// TwinCAT 3 PLC project PLC1
// ProgramVersion: 3.1.4023.0
// libraries:
//   Tc2_Standard, * (Beckhoff Automation GmbH)
//   Tc2_System, * (Beckhoff Automation GmbH)
//   Tc3_Module, * (Beckhoff Automation GmbH)
// project tree:
//   / PlcTask.TcTTO
//   POUs/ MAIN.TcPOU
//   POUs/SD_Valve/ SD_Valve.TcPOU
//   POUs/SD_Valve/States/ InitState.TcPOU, AutoState.TcPOU, ManualState.TcPOU, I_SD_ValveState.TcIO
//   POUs/SD_Valve/Transitions/ GoToManual.TcPOU, GoToInit.TcPOU, GoToAuto.TcPOU, I_Transitive.TcIO
// real-time tasks:
//   TASK PlcTask: cycle T#10ms, priority 20, ADS port 350

CONFIGURATION PLC1
    RESOURCE PLC ON TwinCAT3
        TASK PlcTask(INTERVAL := T#10ms, PRIORITY := 20);
        PROGRAM MAIN WITH PlcTask : MAIN;
    END_RESOURCE
END_CONFIGURATION

// ---- POUs/SD_Valve/States/I_SD_ValveState.TcIO
INTERFACE I_SD_ValveState

METHOD Close : BOOL
VAR_INPUT
END_VAR
END_METHOD

METHOD Open : BOOL
VAR_INPUT
END_VAR
END_METHOD

METHOD RUN
END_METHOD

METHOD SetTransition
VAR_INPUT
    transition : I_Transitive;
END_VAR
END_METHOD

PROPERTY StateName : STRING
GET
END_GET
END_PROPERTY

END_INTERFACE

// ---- POUs/SD_Valve/Transitions/I_Transitive.TcIO
INTERFACE I_Transitive

METHOD Transit
VAR_INPUT
END_VAR
END_METHOD

END_INTERFACE

// ---- POUs/MAIN.TcPOU
PROGRAM MAIN
VAR
    sdValve : SD_Valve;
    openCmd : BOOL;
    openResult : BOOL;
    closeCmd : BOOL;
    closeResult : BOOL;
    goToAutoCmd : BOOL;
    goToManaulCmd : BOOL;
    goToInitCmd : BOOL;
END_VAR

sdValve();

IF openCmd THEN
    openCmd := FALSE;
    openResult := FALSE;
    openResult :=sdValve.OpenValve();
END_IF

IF closeCmd THEN
    closeCmd := FALSE;
    closeResult := FALSE;
    closeResult := sdValve.CloseValve();
END_IF

IF goToAutoCmd THEN
    goToAutoCmd := FALSE;
    sdValve.GoToAutoState();
END_IF

IF goToManaulCmd THEN
    goToManaulCmd := FALSE;
    sdValve.GoToManualState();
END_IF

IF goToInitCmd THEN
    goToInitCmd := FALSE;
    sdValve.GoToInitState();
END_IF

END_PROGRAM

// ---- POUs/SD_Valve/SD_Valve.TcPOU
FUNCTION_BLOCK SD_Valve
VAR_INPUT
END_VAR
VAR_OUTPUT
    coil : BOOL;
END_VAR
VAR
    _initState : InitState(THIS);
    _autoState : AutoState(THIS);
    _manualState : ManualState(THIS);
    _state : I_SD_ValveState := _initState;
    _stateName : STRING;
    _goToInit : GoToInit(ADR(_state), _initState);
    _goToAuto : GoToAuto(ADR(_state), _autoState);
    _goToManual : GoToManual(ADR(_state), _manualState);
    _setDefaultTransitions : BOOL := TRUE;
END_VAR

IF _setDefaultTransitions THEN
    _setDefaultTransitions := FALSE;
    _initState.SetTransition(_goToAuto);
END_IF

_state.RUN();
_stateName := _state.StateName;

METHOD CloseValve : BOOL
CloseValve := _state.Close();
END_METHOD

METHOD GoToAutoState
IF _state.StateName = _autoState.StateName THEN
    RETURN;
END_IF

IF _state.StateName = _initState.StateName THEN
    _state.SetTransition(_goToAuto);
ELSE
    _goToInit.Transit();
END_IF
END_METHOD

METHOD GoToInitState
IF _state.StateName = _initState.StateName THEN
    RETURN;
END_IF

_goToInit.Transit();
END_METHOD

METHOD GoToManualState
IF _state.StateName = _manualState.StateName THEN
    RETURN;
END_IF

IF _state.StateName = _initState.StateName THEN
    _state.SetTransition(_goToManual);
ELSE
    _goToManual.Transit();
END_IF
END_METHOD

METHOD OpenValve : BOOL
OpenValve := _state.Open();
END_METHOD

END_FUNCTION_BLOCK

// ---- POUs/SD_Valve/States/InitState.TcPOU
FUNCTION_BLOCK InitState IMPLEMENTS I_SD_ValveState
VAR_INPUT
END_VAR
VAR_OUTPUT
END_VAR
VAR
    _ptSdValve : POINTER TO SD_Valve;
    _transition : I_Transitive;
    delayTimer : Tc2_Standard.TON;
    start : BOOL;
END_VAR

delayTimer(IN:=start,PT:=T#10S);
IF NOT start THEN
    start := TRUE;
END_IF
IF delayTimer.q THEN
    start := FALSE;
//    _ptSdValve^.GoToAutoState();
    IF _transition<>0 THEN
        _transition.Transit();
	END_IF
END_IF

METHOD Close : BOOL
Close := false;
END_METHOD

METHOD FB_init : BOOL
VAR_INPUT
	bInitRetains : BOOL; // if TRUE, the retain variables are initialized (warm start / cold start)
	bInCopyCode : BOOL;  // if TRUE, the instance afterwards gets moved into the copy code (online change)
    ptSdValve : POINTER TO SD_Valve;
END_VAR
_ptSdValve := ptSdValve;
END_METHOD

METHOD Open : BOOL
Open := False;
END_METHOD

METHOD RUN
THIS^();
END_METHOD

METHOD SetTransition
VAR_INPUT
	transition	: I_Transitive;
END_VAR
_transition := transition;
END_METHOD

PROPERTY StateName : STRING
GET
StateName := 'Init';
END_GET
END_PROPERTY

END_FUNCTION_BLOCK

// ---- POUs/SD_Valve/States/AutoState.TcPOU
FUNCTION_BLOCK AutoState IMPLEMENTS I_SD_ValveState
VAR_INPUT
END_VAR
VAR_OUTPUT
END_VAR
VAR
    _ptSdValve : POINTER TO SD_Valve;
    _transition : I_Transitive;
END_VAR

METHOD Close : BOOL
Close := TRUE;
END_METHOD

METHOD FB_init : BOOL
VAR_INPUT
	bInitRetains : BOOL; // if TRUE, the retain variables are initialized (warm start / cold start)
	bInCopyCode : BOOL;  // if TRUE, the instance afterwards gets moved into the copy code (online change)
    ptSdValve : POINTER TO SD_Valve;
END_VAR
_ptSdValve := ptSdValve;
END_METHOD

METHOD Open : BOOL
Open := true;
END_METHOD

METHOD RUN
THIS^();
END_METHOD

METHOD SetTransition
VAR_INPUT
	transition	: I_Transitive;
END_VAR
_transition := transition;
END_METHOD

PROPERTY StateName : STRING
GET
StateName := 'Auto';
END_GET
END_PROPERTY

END_FUNCTION_BLOCK

// ---- POUs/SD_Valve/States/ManualState.TcPOU
FUNCTION_BLOCK ManualState IMPLEMENTS I_SD_ValveState
VAR_INPUT
END_VAR
VAR_OUTPUT
END_VAR
VAR
    _ptSdValve : POINTER TO SD_Valve;
    _transition : I_Transitive;
    delayTimer : Tc2_Standard.TP;
    command : BOOL;
END_VAR

delayTimer(IN:=command,PT:=T#5S);
IF command THEN
    command := FALSE;
END_IF

METHOD Close : BOOL
IF delayTimer.Q THEN
    Close := FALSE;
ELSE
    command := TRUE;
    Close := TRUE;
END_IF
END_METHOD

METHOD FB_init : BOOL
VAR_INPUT
	bInitRetains : BOOL; // if TRUE, the retain variables are initialized (warm start / cold start)
	bInCopyCode : BOOL;  // if TRUE, the instance afterwards gets moved into the copy code (online change)
    ptSdValve : POINTER TO SD_Valve;
END_VAR
_ptSdValve := ptSdValve;
END_METHOD

METHOD Open : BOOL
IF delayTimer.Q THEN
    Open := FALSE;
ELSE
    command := TRUE;
    Open := TRUE;
END_IF
END_METHOD

METHOD RUN
THIS^();
END_METHOD

METHOD SetTransition
VAR_INPUT
	transition	: I_Transitive;
END_VAR
_transition := transition;
END_METHOD

PROPERTY StateName : STRING
GET
StateName := 'Manual';
END_GET
END_PROPERTY

END_FUNCTION_BLOCK

// ---- POUs/SD_Valve/Transitions/GoToInit.TcPOU
FUNCTION_BLOCK GoToInit IMPLEMENTS I_Transitive
VAR
    _currentState : POINTER TO I_SD_ValveState;
    _nextState : REFERENCE TO InitState;
END_VAR

METHOD FB_init : BOOL
VAR_INPUT
	bInitRetains : BOOL; // if TRUE, the retain variables are initialized (warm start / cold start)
	bInCopyCode : BOOL;  // if TRUE, the instance afterwards gets moved into the copy code (online change)
    currentState : POINTER TO I_SD_ValveState;
    nextState : REFERENCE TO InitState;
END_VAR
_currentState := currentState;
_nextState REF= nextState;
END_METHOD

METHOD Transit
_currentState^ := _nextState;
END_METHOD

END_FUNCTION_BLOCK

// ---- POUs/SD_Valve/Transitions/GoToAuto.TcPOU
FUNCTION_BLOCK GoToAuto IMPLEMENTS I_Transitive
VAR
    _currentState : POINTER TO I_SD_ValveState;
    _nextState : REFERENCE TO AutoState;
END_VAR

METHOD FB_init : BOOL
VAR_INPUT
	bInitRetains : BOOL; // if TRUE, the retain variables are initialized (warm start / cold start)
	bInCopyCode : BOOL;  // if TRUE, the instance afterwards gets moved into the copy code (online change)
    currentState : POINTER TO I_SD_ValveState;
    nextState : REFERENCE TO AutoState;
END_VAR
_currentState := currentState;
_nextState REF= nextState;
END_METHOD

METHOD Transit
_currentState^ := _nextState;
END_METHOD

END_FUNCTION_BLOCK

// ---- POUs/SD_Valve/Transitions/GoToManual.TcPOU
FUNCTION_BLOCK GoToManual IMPLEMENTS I_Transitive
VAR
    _currentState : POINTER TO I_SD_ValveState;
    _nextState : REFERENCE TO ManualState;
END_VAR

METHOD FB_init : BOOL
VAR_INPUT
	bInitRetains : BOOL; // if TRUE, the retain variables are initialized (warm start / cold start)
	bInCopyCode : BOOL;  // if TRUE, the instance afterwards gets moved into the copy code (online change)
    currentState : POINTER TO I_SD_ValveState;
    nextState : REFERENCE TO ManualState;
END_VAR
_currentState := currentState;
_nextState REF= nextState;
END_METHOD

METHOD Transit
_currentState^ := _nextState;
END_METHOD

END_FUNCTION_BLOCK
